TYPE PathHandle_t : Pointer to StrFileName_t; END_TYPE

(* stored: Version 1.1.0.1, ProductVersion 3.1.4024.12
   DUT PathHandle_t: Id {f09e1a23-dbcc-42ce-b40d-d91eb277be2c} *)
